TYPE T_PROCESS : WORD; END_TYPE

(* stored: Version 1.1.0.1
   DUT T_PROCESS: Id {75be7743-921f-40fe-964e-75835d4f2662} *)
